PROGRAM USB
VAR
END_VAR

;

END_PROGRAM

(* stored: Version 1.1.0.1, ProductVersion 3.1.0.26
   POU USB: Id {0aa25fed-cd14-47ae-a3b5-a6d0f8d7d19f} *)
